FUNCTION_BLOCK FB 49
TITLE = 'flour_fault_faults'
AUTHOR : CB


VAR_INPUT
	generalFault3 : BOOL := FALSE;	//Défaut général
	generalFault2 : BOOL := FALSE;	//Défaut général
	generalFault1 : BOOL := FALSE;	//Défaut général
END_VAR

VAR_OUTPUT
	fault : BOOL := FALSE;	//
END_VAR

BEGIN


NETWORK
TITLE =
//
L1:	O	generalFault3;
O	generalFault1;
O	generalFault2;
=	fault;




NETWORK
TITLE =
//
L2:	NOP 0



NETWORK
TITLE =
//
L3:	NOP 0




END_FUNCTION_BLOCK
